FUNCTION_BLOCK Wago1504_5 (* Service Interface Function Block Type *)
  (* Standard: 61499-2; Description: Copyright (c) 2018 fortiss GmbH This program and the accompanying materials are made available under the terms of the Eclipse Public License 2.0 which is available at https://www.eclipse.org/legal/epl-2.0/ SPDX-License-Identifier: EPL-2.0 *)
  (* Version 1.0, 2018-12-05, Jose Cabral *)
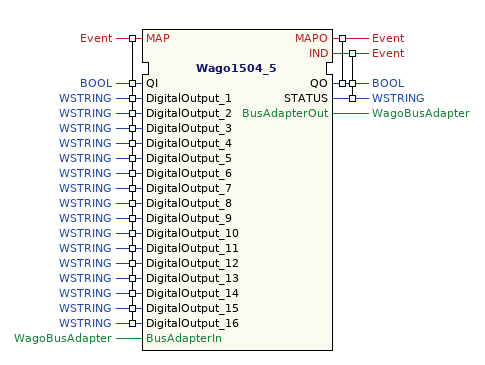
  EVENT_INPUT
    MAP WITH DigitalOutput_1, DigitalOutput_2, DigitalOutput_5, DigitalOutput_3, DigitalOutput_4, DigitalOutput_6, DigitalOutput_7, DigitalOutput_8, DigitalOutput_9, DigitalOutput_10, DigitalOutput_11, DigitalOutput_12, DigitalOutput_13, DigitalOutput_14, DigitalOutput_15, DigitalOutput_16, QI; (* Map Pins *)
  END_EVENT
  EVENT_OUTPUT
    MAPO WITH QO; (* Confirm Pin Mapping *)
    IND WITH QO, STATUS; (* Indication from Resource *)
  END_EVENT
  VAR_INPUT
    QI : BOOL; (* Event Input Qualifier *)
    DigitalOutput_1 : WSTRING;
    DigitalOutput_2 : WSTRING;
    DigitalOutput_3 : WSTRING;
    DigitalOutput_4 : WSTRING;
    DigitalOutput_5 : WSTRING;
    DigitalOutput_6 : WSTRING;
    DigitalOutput_7 : WSTRING;
    DigitalOutput_8 : WSTRING;
    DigitalOutput_9 : WSTRING;
    DigitalOutput_10 : WSTRING;
    DigitalOutput_11 : WSTRING;
    DigitalOutput_12 : WSTRING;
    DigitalOutput_13 : WSTRING;
    DigitalOutput_14 : WSTRING;
    DigitalOutput_15 : WSTRING;
    DigitalOutput_16 : WSTRING;
  END_VAR
  VAR_OUTPUT
    QO : BOOL; (* Event Output Qualifier *)
    STATUS : WSTRING; (* Service Status *)
  END_VAR
  SOCKETS
    BusAdapterIn : WagoBusAdapter;
  END_SOCKETS
  PLUGS
    BusAdapterOut : WagoBusAdapter;
  END_PLUGS
END_FUNCTION_BLOCK
